{attribute 'GeneratedUsingTerminal: EK1100-0000-0018'}
{attribute addProperty BoxType "EK1100-0000-0018"}
{attribute addProperty Id "Beckhoff_ER2xxxEK1122Beckhoff_ER2xxxEK1122_1CCCDC5A910"}
{attribute addProperty CRC "1150381965"}
{attribute addProperty Size "910"}
TYPE Beckhoff_ER2xxx_44916F8D EXTENDS EK1100_AB5A9467 :
STRUCT
	{attribute addProperty Name "Beckhoff_ER2xxxEK1122"}
	{attribute addProperty PreviousPort "Beckhoff ER2xxx : B"}
	Beckhoff_ER2xxxEK1122 : Beckhoff_ER2xxxEK1122_1CCCDC5A;
END_STRUCT
END_TYPE

(* stored: Version 1.2.0.0, ProductVersion 3.1.4024.9
   DUT Beckhoff_ER2xxx_44916F8D: Id {d6a1698d-91c0-4be3-b424-9fad9c10f0d6} *)
